// TIA Portal V19 export
DATA_BLOCK "DEBUG_MES_Receive_Msg_Topic4XX"   // DB206
// stored: MemoryReserve 100
   VAR
      DEBUG_RECEIVE : Struct
         Enable : Bool;
         AckChangeStep : Bool;
         ActualStep : Int;
      END_STRUCT;
      ACK_MSG_enable : Bool;
      NEW_MSG_401 : Struct   // Invio dati rotolo aspo in carico
         ABILITA_FC : Bool;
         EXE_MSG : Bool;
         MSG : "MES_Msg";
      END_STRUCT;
      NEW_MSG_402 : Struct   // Rimozioni dati rotolo aspo in carico
         ABILITA_FC : Bool;
         EXE_MSG : Bool;
         MSG : "MES_Msg";
      END_STRUCT;
      NEW_MSG_403 : Struct   // Richiesta ulteriore provino
         ABILITA_FC : Bool;
         EXE_MSG : Bool;
         MSG : "MES_Msg";
      END_STRUCT;
      NEW_MSG_410 : Struct   // Interrogazione stato rotolo aspo in linea
         ABILITA_FC : Bool;
         EXE_MSG : Bool;
         MSG : "MES_Msg";
      END_STRUCT;
      NEW_MSG_412 : Struct   // Interrogazione stato rotolo aspo in carico
         ABILITA_FC : Bool;
         EXE_MSG : Bool;
         MSG : "MES_Msg";
      END_STRUCT;
      NEW_MSG_422 : Struct   // Interrogazione stato rotolo taglio finale
         ABILITA_FC : Bool;
         EXE_MSG : Bool;
         MSG : "MES_Msg";
      END_STRUCT;
   END_VAR
BEGIN
END_DATA_BLOCK
